// LS Electric XG5000 project: 동남145
// PLC NewPLC
// module base 0 slot 0: 입출력 모듈:XBC-DN/DP14E (DC 24V 입력 8점, 트랜지스터 출력 6점)

PROGRAM NewProgram (task: 스캔 프로그램)

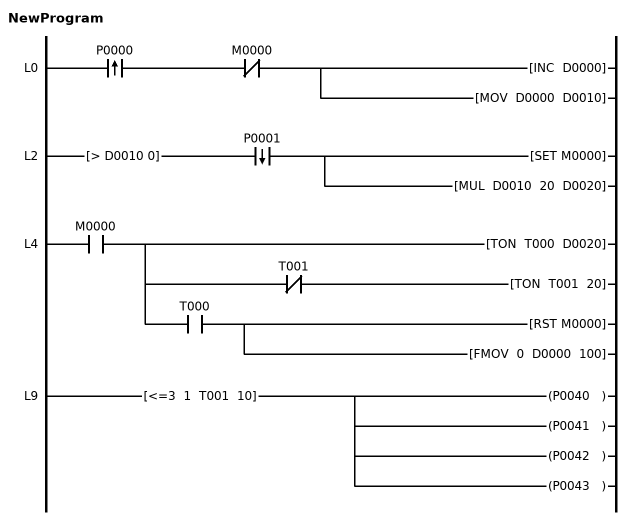
; L0
LOADP     P0000
AND NOT   M0000
INC       D0000
MOV       D0000 D0010
; L2
LOAD>     D0010 0
ANDN      P0001
SET       M0000
MUL       D0010 20 D0020
; L4
LOAD      M0000
TON       T000 D0020
MPUSH
AND NOT   T001
TON       T001 20
MPOP
AND       T000
RST       M0000
FMOV      0 D0000 100
; L9
LOAD<=3   1 T001 10
OUT       P0040
OUT       P0041
OUT       P0042
OUT       P0043